PROGRAM MAIN
VAR
	StopRichiesto: BOOL;
	Anomalia: BOOL;
	Emergenza: BOOL;
	OperazioneInCorso: BOOL;
	Funzione: BOOL;
	Smistamento: BOOL;
	Rotazione: BOOL;
	AttivaMicroRulli: BOOL;
	FineSmistamento: BOOL;
	FinePesatura: BOOL;
	RuotaOrigine: BOOL;
	PesoMin5: BOOL;
	PesoMag10: BOOL;
	PesoIntermedio: BOOL;
	ProsciuttoSmistato: BOOL;
	ProsciuttiTotali: UINT;
	ProsciuttiCommerciabili: UINT;
	PercentualeProsciuttiCommerciabili: UINT;
	//Timer
	TON_PS1: TON;
	TON_Pesatura: TON;
	TON_MicroRulli: TON;
	//Counter
	CTU_Min5: CTU;
	CTU_Mag10: CTU;
	CTU_Intermedi: CTU;
	AttivaPistone: BOOL;
	PezzoBianco: BOOL;
	PezzoNero: BOOL;
	SpostaTrapano: BOOL;
	AttivaBlocco: BOOL;
	AttivaTrapano: BOOL;
	AttivaTimbratura: BOOL;
	TON_Pistone: TON;
	Foratura: BOOL;
	Timbratura: BOOL;
END_VAR
VAR // added by the converter: edge detectors and wires of the graphical bodies
    _w1 : BOOL;
END_VAR

GestionePulsanti();
GestioneMotori();
GestioneSmistamento();

ACTION GestioneConteggio:
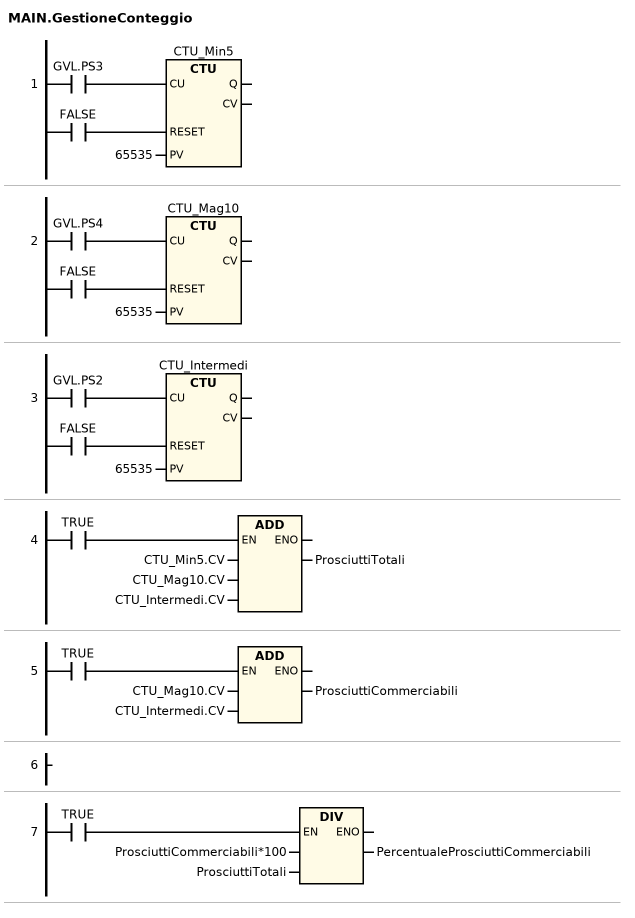
// NETWORK 1
CTU_Min5(CU := GVL.PS3, RESET := FALSE, PV := 65535); // CTU

// NETWORK 2
CTU_Mag10(CU := GVL.PS4, RESET := FALSE, PV := 65535); // CTU

// NETWORK 3
CTU_Intermedi(CU := GVL.PS2, RESET := FALSE, PV := 65535); // CTU

// NETWORK 4
ProsciuttiTotali := CTU_Min5.CV + CTU_Mag10.CV + CTU_Intermedi.CV;

// NETWORK 5
ProsciuttiCommerciabili := CTU_Mag10.CV + CTU_Intermedi.CV;

// NETWORK 6

// NETWORK 7
PercentualeProsciuttiCommerciabili := (ProsciuttiCommerciabili*100) / ProsciuttiTotali;
END_ACTION

ACTION GestioneMotori:
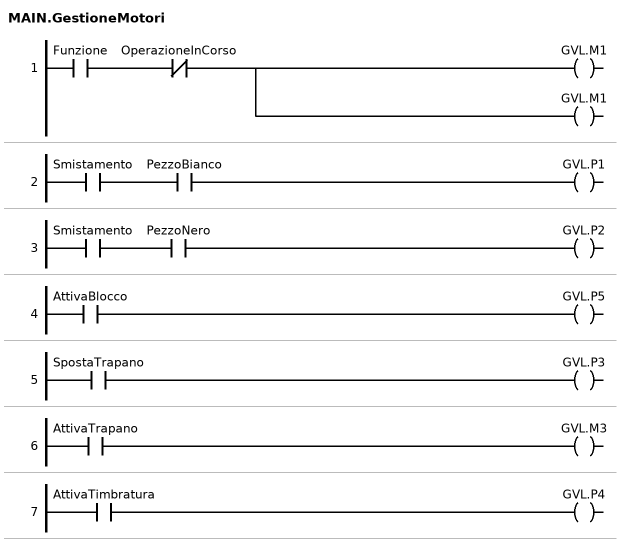
// NETWORK 1
_w1 := Funzione AND NOT OperazioneInCorso;
GVL.M1 := _w1;
GVL.M1 := _w1;

// NETWORK 2
GVL.P1 := Smistamento AND PezzoBianco;

// NETWORK 3
GVL.P2 := Smistamento AND PezzoNero;

// NETWORK 4
GVL.P5 := AttivaBlocco;

// NETWORK 5
GVL.P3 := SpostaTrapano;

// NETWORK 6
GVL.M3 := AttivaTrapano;

// NETWORK 7
GVL.P4 := AttivaTimbratura;
END_ACTION

ACTION GestionePulsanti:
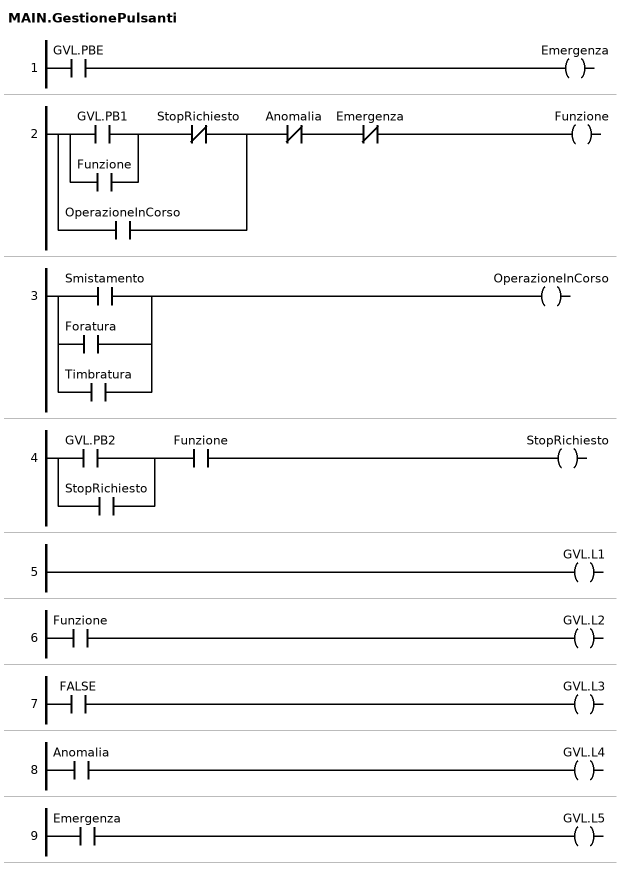
// NETWORK 1
Emergenza := GVL.PBE;

// NETWORK 2
Funzione := ((GVL.PB1 OR Funzione) AND NOT StopRichiesto OR OperazioneInCorso) AND NOT Anomalia AND NOT Emergenza;

// NETWORK 3
OperazioneInCorso := Smistamento OR Foratura OR Timbratura;

// NETWORK 4
StopRichiesto := (GVL.PB2 OR StopRichiesto) AND Funzione;

// NETWORK 5
GVL.L1 := TRUE;

// NETWORK 6
GVL.L2 := Funzione;

// NETWORK 7
GVL.L3 := FALSE;

// NETWORK 8
GVL.L4 := Anomalia;

// NETWORK 9
GVL.L5 := Emergenza;
END_ACTION

ACTION GestioneRotazione:
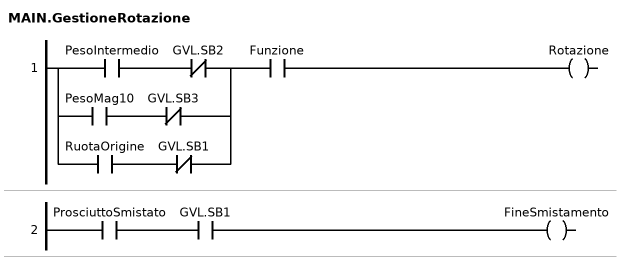
// NETWORK 1
Rotazione := (PesoIntermedio AND NOT GVL.SB2 OR PesoMag10 AND NOT GVL.SB3 OR RuotaOrigine AND NOT GVL.SB1) AND Funzione;

// NETWORK 2
FineSmistamento := ProsciuttoSmistato AND GVL.SB1;
END_ACTION

ACTION GestioneSmistamento:
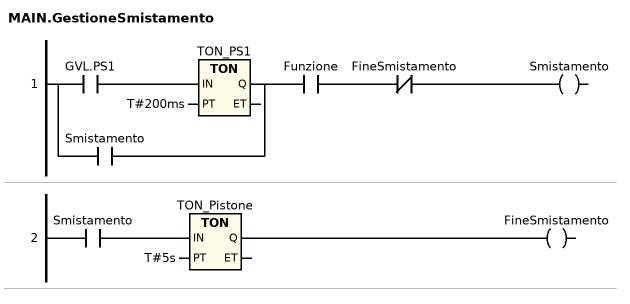
// NETWORK 1
TON_PS1(IN := GVL.PS1, PT := T#200ms); // TON
Smistamento := (TON_PS1.Q OR Smistamento) AND Funzione AND NOT FineSmistamento;

// NETWORK 2
TON_Pistone(IN := Smistamento, PT := T#5s); // TON
FineSmistamento := TON_Pistone.Q;
END_ACTION

ACTION GestioneSmistamento2:
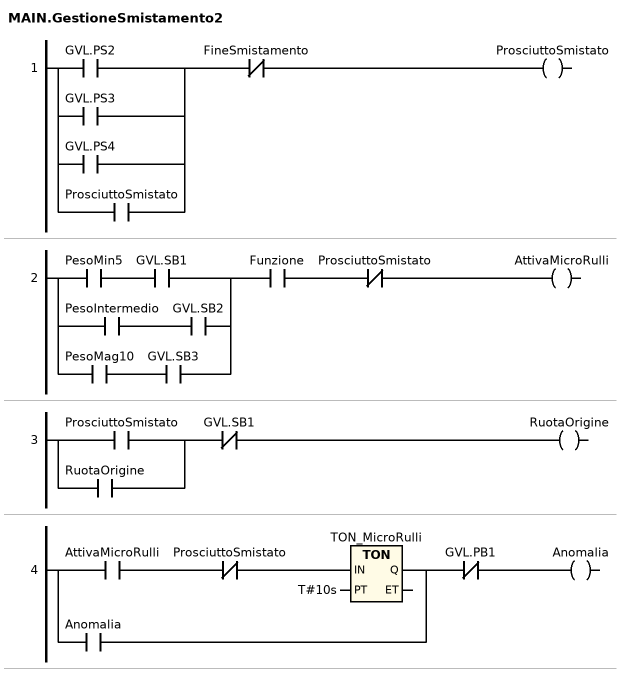
// NETWORK 1
ProsciuttoSmistato := (GVL.PS2 OR GVL.PS3 OR GVL.PS4 OR ProsciuttoSmistato) AND NOT FineSmistamento;

// NETWORK 2
AttivaMicroRulli := (PesoMin5 AND GVL.SB1 OR PesoIntermedio AND GVL.SB2 OR PesoMag10 AND GVL.SB3) AND Funzione AND NOT ProsciuttoSmistato;

// NETWORK 3
RuotaOrigine := (ProsciuttoSmistato OR RuotaOrigine) AND NOT GVL.SB1;

// NETWORK 4
TON_MicroRulli(IN := AttivaMicroRulli AND NOT ProsciuttoSmistato, PT := T#10s); // TON
Anomalia := (TON_MicroRulli.Q OR Anomalia) AND NOT GVL.PB1;
END_ACTION

END_PROGRAM

(* stored: Version 1.1.0.1, ProductVersion 3.1.4024.12
   POU MAIN: Id {77ce3c58-9155-42f5-9eb6-c02febfddbf9}, SpecialFunc None
   Action GestioneConteggio: Id {6d95f27d-0282-4140-898e-f4ab137f763b}
   Action GestioneMotori: Id {90fd2a52-73a3-4857-abe4-70f7165621aa}
   Action GestionePulsanti: Id {3f00a759-f8d0-455e-af78-03f29b3994ec}
   Action GestioneRotazione: Id {dcd47c17-31b5-470b-b8df-fa6a694df16f}
   Action GestioneSmistamento: Id {afcac87d-3588-48ef-84da-e3c3b38ed934}
   Action GestioneSmistamento2: Id {6af05be5-420f-47a5-a7ce-bdc4d670b5af} *)
